FUNCTION_BLOCK ErrorTest
VAR_INPUT
END_VAR
VAR_OUTPUT
END_VAR
VAR
	EventLoggerMessage : FB_TcMessage;
	bInit : bool := false;
END_VAR

IF bInit = FALSE THEN
	bInit := TRUE;
	EventLoggerMessage.CreateEx(TC_EVENTS.Events.TestEvent, 0);
END_IF

EventLoggerMessage.Send(0);

END_FUNCTION_BLOCK

(* stored: Version 1.1.0.1
   POU ErrorTest: Id {97fd7844-39ed-4856-92b7-76b406dfb6f1}, SpecialFunc None *)
